// TIA Portal V20 export
DATA_BLOCK "SBK06"   // DB202
// stored: MemoryReserve 100
   VAR
      "GATE EC U/W BTM PB.LOCK" : Bool := FALSE;
      "GATE EC U/W BTM PB.RESET" : Bool := FALSE;
      SPARE : Bool := FALSE;
      SPARE_1 : Bool := FALSE;
      "GATE EC U/W BTM PB.UNLOCK" : Bool := FALSE;
      SPARE_2 : Bool := FALSE;
      SPARE_3 : Bool := FALSE;
      SPARE_4 : Bool := FALSE;
      "GATE EC U/W BTM PL.LOCK" : Bool := TRUE;
      "GATE EC U/W BTM PL.UNLOCK" : Bool := TRUE;
      "GATE EC U/W BTM PL.RESET" : Bool := TRUE;
   END_VAR
BEGIN
END_DATA_BLOCK
